PROGRAM VisuInit
VAR
END_VAR

gHMIData.gVisuHasInited := TRUE;

END_PROGRAM

(* stored: Version 1.1.0.1, ProductVersion 3.1.4024.11
   POU VisuInit: Id {33320dae-9040-0cbf-1fe5-5e8fdd99e2f4}, SpecialFunc None *)
